// TIA Portal V19 export
ORGANIZATION_BLOCK "Main"   // OB1, LAD, ProgramCycle
TITLE = "Main Program Sweep (Cycle)"
{ S7_Optimized_Access := 'TRUE' }
// stored: SetENOAutomatically false
   VAR_INPUT
      Initial_Call : Bool;   // Initial call of this OB
      Remanence : Bool;   // =True, if remanent data are available
   END_VAR
BEGIN

REGION Network 1
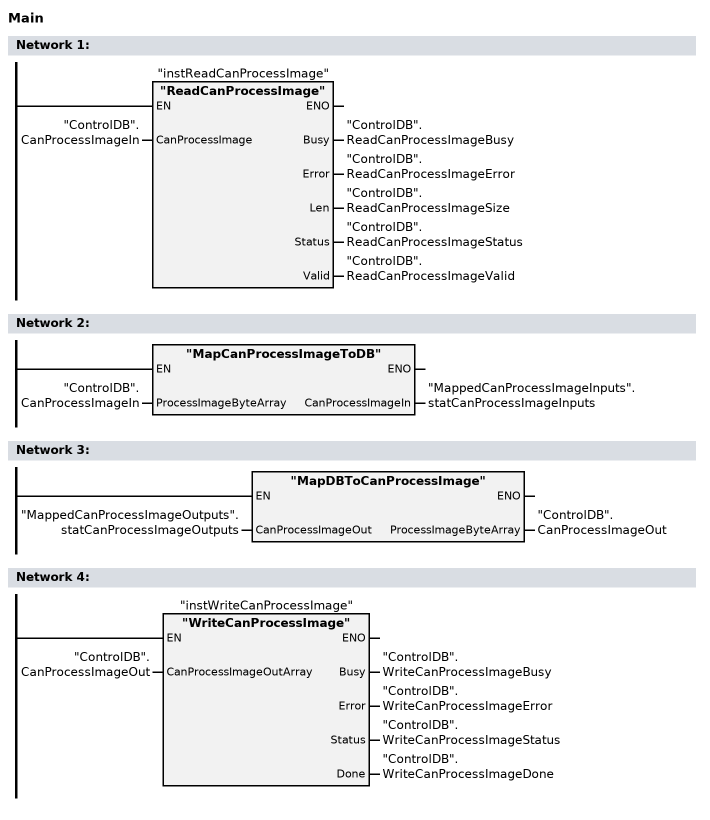
   RUNG wire#powerrail
      "instReadCanProcessImage"(CanProcessImage := "ControlDB".CanProcessImageIn, Busy => "ControlDB".ReadCanProcessImageBusy, Error => "ControlDB".ReadCanProcessImageError, Len => "ControlDB".ReadCanProcessImageSize, Status => "ControlDB".ReadCanProcessImageStatus, Valid => "ControlDB".ReadCanProcessImageValid)
   END_RUNG
   // the same network as SCL:
   "instReadCanProcessImage"(CanProcessImage := "ControlDB".CanProcessImageIn,   // "ReadCanProcessImage"
                           Busy => "ControlDB".ReadCanProcessImageBusy,
                           Error => "ControlDB".ReadCanProcessImageError,
                           Len => "ControlDB".ReadCanProcessImageSize,
                           Status => "ControlDB".ReadCanProcessImageStatus,
                           Valid => "ControlDB".ReadCanProcessImageValid);
END_REGION

REGION Network 2
   RUNG wire#powerrail
      "MapCanProcessImageToDB"(ProcessImageByteArray := "ControlDB".CanProcessImageIn, CanProcessImageIn => "MappedCanProcessImageInputs".statCanProcessImageInputs)
   END_RUNG
   // the same network as SCL:
   "MapCanProcessImageToDB"(ProcessImageByteArray := "ControlDB".CanProcessImageIn,
                           CanProcessImageIn => "MappedCanProcessImageInputs".statCanProcessImageInputs);
END_REGION

REGION Network 3
   RUNG wire#powerrail
      "MapDBToCanProcessImage"(CanProcessImageOut := "MappedCanProcessImageOutputs".statCanProcessImageOutputs, ProcessImageByteArray => "ControlDB".CanProcessImageOut)
   END_RUNG
   // the same network as SCL:
   "MapDBToCanProcessImage"(CanProcessImageOut := "MappedCanProcessImageOutputs".statCanProcessImageOutputs,
                           ProcessImageByteArray => "ControlDB".CanProcessImageOut);
END_REGION

REGION Network 4
   RUNG wire#powerrail
      "instWriteCanProcessImage"(CanProcessImageOutArray := "ControlDB".CanProcessImageOut, Busy => "ControlDB".WriteCanProcessImageBusy, Error => "ControlDB".WriteCanProcessImageError, Status => "ControlDB".WriteCanProcessImageStatus, Done => "ControlDB".WriteCanProcessImageDone)
   END_RUNG
   // the same network as SCL:
   "instWriteCanProcessImage"(CanProcessImageOutArray := "ControlDB".CanProcessImageOut,   // "WriteCanProcessImage"
                           Busy => "ControlDB".WriteCanProcessImageBusy,
                           Error => "ControlDB".WriteCanProcessImageError,
                           Status => "ControlDB".WriteCanProcessImageStatus,
                           Done => "ControlDB".WriteCanProcessImageDone);
END_REGION
END_ORGANIZATION_BLOCK
